Staubli VAL3: isLatched.pgx

public program isLatched(bool& x_bLatched[] (dimensions=1))
begin
  // This program checks if the number of latch for
  // the part detection has been reached
  //
  //
  // Output Param
  // x_bLatched  : If true, a part has been detected
  //
  //----------------------------------------------------------------
  //
  if bPartLatched==true
    x_bLatched=true
  else
    x_bLatched=false
  endIf
end
